FUNCTION_BLOCK FB_Blinker
VAR_INPUT
	bStart: BOOL;
	tSignalTimeOn: TIME;
	tSignalTimeOff: TIME;
END_VAR
VAR_OUTPUT
	bOut: BOOL;
END_VAR
VAR
	fbTimerA: TON;
	fbTimerB: TON;
END_VAR

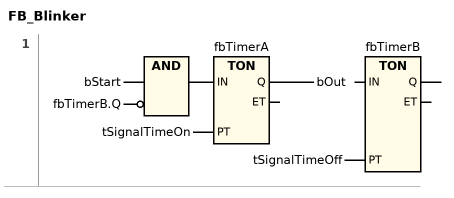
// NETWORK 1
fbTimerA(IN := bStart AND NOT fbTimerB.Q, PT := tSignalTimeOn); // TON
bOut := fbTimerA.Q;
fbTimerB(IN := fbTimerA.Q, PT := tSignalTimeOff); // TON

END_FUNCTION_BLOCK

(* stored: Version 1.1.0.1, ProductVersion 3.1.4024.4
   POU FB_Blinker: Id {edbc8775-ccfe-4b93-8176-dd79d7288f41}, SpecialFunc None *)
